TYPE T_PBC_DATACHN :
STRUCT
	rSendData: T_IdBaseSendData;
END_STRUCT
END_TYPE

(* stored: Version 1.1.0.1, ProductVersion 3.1.0.36
   DUT T_PBC_DATACHN: Id {b01a29ff-b50f-47fc-9b52-ea331b9e8cd3} *)
